(* PLC project v0.6.02_RefactorGateAndTest.project, CODESYS CODESYS V3.5 SP19 Patch 1 *)
(* stored: creationDateTime 2026-08-11T14:02:33.676658, modificationDateTime 2026-08-11T14:02:33.676658 *)

(* ═══════════════════════════════════════════════════════════════ 🎮 ST_DredgingAssistCmd — Sélections IHM assistance prélèvement ═══════════════════════════════════════════════════════════════ *)
TYPE ST_DredgingAssistCmd : STRUCT
  TglEnableDiveSearch : BOOL := TRUE;  (* Assistance plongée active *)
  TglEnableExtractionSequence : BOOL := TRUE;  (* Assistance extraction active *)
  TglBucketAtBottomConfirmed : BOOL := FALSE;  (* Attestation manuelle temporaire du fond *)
  TglBypassDiveSearchSequence : BOOL := FALSE;  (* 🆕 2026-08-07 (9) : bypass simplifié de la séquence FB_DiveSearch complète (préconditions strictes -- benne ouverte, DiveStartMin_M, fenêtre immersion). Si TRUE, un front MONTANT Kobold pendant une descente confirme directement le fond, sans passer par l'état-machine FB_DiveSearch (qui continue de tourner en parallèle, inchangée -- utile pour KoboldMeasureEnable). Défaut FALSE : comportement identique à avant (séquence complète seule source de confirmation). *)
  TglEnableDumpAtTremie : BOOL := TRUE;  (* 🆕 2026-08-07 : mode vidage à la trémie — *)
END_STRUCT;
END_TYPE
